// TIA Portal V18 export
DATA_BLOCK "_DOOORS"   // DB71
VERSION : 0.1
// stored: AutoNumber true, DBAccessibleFromOPCUA true, InstanceOfName _DOOORS_fb, InstanceOfType FB
"_DOOORS_fb"
   // VAR_INPUT
   //    xBtnOpen : Bool;
   //    xBtnClose : Bool;
   //    allowedNotAuto : Bool;
   //    allowedCloseLightBrrier : Bool;
   //    allowedCloseManipulator : Bool;
   //    xClosed : Bool;
   //    xOpen : Bool;
   // END_VAR
   // VAR_OUTPUT
   //    yCmdOpen : Bool;
   //    yCmdClose : Bool;
   //    sOpen : Bool;
   //    sClosed : Bool;
   //    wn_Auto : Bool;
   //    wnLightbarrier : Bool;
   //    wnManipulatorClose : Bool;
   // END_VAR
   // VAR_IN_OUT
   //    yBeepCosedResetMe : Bool;
   // END_VAR
   // VAR
   //    memOpen : Bool;
   //    memClosed : Bool;
   //    memopn : Bool;
   //    memopn1 : Bool;
   //    memClosed1 : Bool;
   // END_VAR
BEGIN
END_DATA_BLOCK
